PROGRAM G7_General
VAR_INPUT	SFCInit:BOOL;	END_VAR
VAR
	Memo_X_Precedent	:LREAL;	//Si plusieurs usinages au même X, pas besoin d'ouvrir et dég à chaque fois 
	Top_Cycles_Palp_Laser	:BOOL; //Lance le G7 des palpages buse et sommet du laser
	Fb_decode_real_Fct_M_: Fb_decode_real;
	Num_Unite_Cycle_Auto: INT;
	Num_operation_Cycle: INT;
	
	FE_Prepa_ISO_3D, FE_ISO_en_cours: F_trig;
	TON_ISO_en_cours, TON_Fin_Decoupe	:Ton;
	

END_VAR

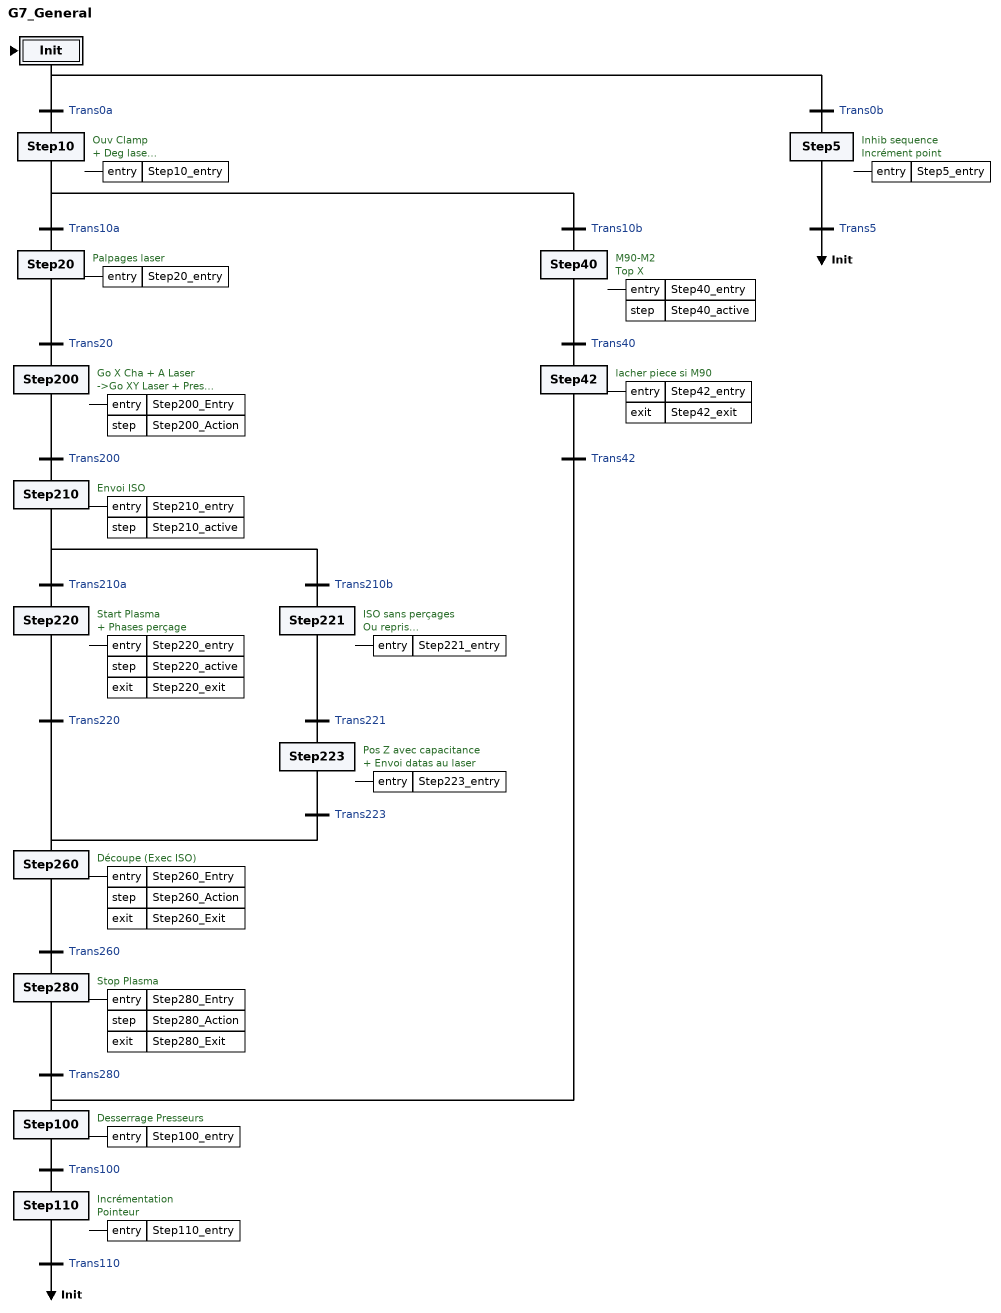
INITIAL_STEP Init:
END_STEP
TRANSITION FROM Init TO Step10
    := Trans0a;
END_TRANSITION
TRANSITION FROM Init TO Step5
    := Trans0b;
END_TRANSITION
// Inhib sequence
// Incrément point
STEP Step5:
    Step5_entry(P1);  // entry action
END_STEP
TRANSITION FROM Step5 TO Init
    := Trans5;
END_TRANSITION
// Ouv Clamp
// + Deg laser
// Si X Diff
// +Ctrl Palp Sommet
STEP Step10:
    Step10_entry(P1);  // entry action
END_STEP
TRANSITION FROM Step10 TO Step20
    := Trans10a;
END_TRANSITION
// Palpages laser
STEP Step20:
    Step20_entry(P1);  // entry action
END_STEP
TRANSITION FROM Step20 TO Step200
    := Trans20;
END_TRANSITION
// Go X Cha + A Laser
// ->Go XY Laser + Press
// +Prépa ISO
STEP Step200:
    Step200_Entry(P1);  // entry action
    Step200_Action(N);  // step action
END_STEP
TRANSITION FROM Step200 TO Step210
    := Trans200;
END_TRANSITION
// Envoi ISO
STEP Step210:
    Step210_entry(P1);  // entry action
    Step210_active(N);  // step action
END_STEP
TRANSITION FROM Step210 TO Step220
    := Trans210a;
END_TRANSITION
// Start Plasma
// + Phases perçage
STEP Step220:
    Step220_entry(P1);  // entry action
    Step220_active(N);  // step action
    Step220_exit(P0);  // exit action
END_STEP
TRANSITION FROM Step220 TO Step260
    := Trans220;
END_TRANSITION
TRANSITION FROM Step210 TO Step221
    := Trans210b;
END_TRANSITION
// ISO sans perçages
// Ou reprise
// Approche rapide Z laser
STEP Step221:
    Step221_entry(P1);  // entry action
END_STEP
TRANSITION FROM Step221 TO Step223
    := Trans221;
END_TRANSITION
// Pos Z avec capacitance
// + Envoi datas au laser
STEP Step223:
    Step223_entry(P1);  // entry action
END_STEP
TRANSITION FROM Step223 TO Step260
    := Trans223;
END_TRANSITION
// Découpe (Exec ISO)
STEP Step260:
    Step260_Entry(P1);  // entry action
    Step260_Action(N);  // step action
    Step260_Exit(P0);  // exit action
END_STEP
TRANSITION FROM Step260 TO Step280
    := Trans260;
END_TRANSITION
// Stop Plasma
STEP Step280:
    Step280_Entry(P1);  // entry action
    Step280_Action(N);  // step action
    Step280_Exit(P0);  // exit action
END_STEP
TRANSITION FROM Step280 TO Step100
    := Trans280;
END_TRANSITION
TRANSITION FROM Step10 TO Step40
    := Trans10b;
END_TRANSITION
// M90-M2
// Top X
STEP Step40:
    Step40_entry(P1);  // entry action
    Step40_active(N);  // step action
END_STEP
TRANSITION FROM Step40 TO Step42
    := Trans40;
END_TRANSITION
// lacher piece si M90
STEP Step42:
    Step42_entry(P1);  // entry action
    Step42_exit(P0);  // exit action
END_STEP
TRANSITION FROM Step42 TO Step100
    := Trans42;
END_TRANSITION
// Desserrage Presseurs
STEP Step100:
    Step100_entry(P1);  // entry action
END_STEP
TRANSITION FROM Step100 TO Step110
    := Trans100;
END_TRANSITION
// Incrémentation
// Pointeur
STEP Step110:
    Step110_entry(P1);  // entry action
END_STEP
TRANSITION FROM Step110 TO Init
    := Trans110;
END_TRANSITION

TRANSITION _tTrans210_1:
FE_Prepa_ISO_3D.Q
END_TRANSITION

ACTION Step10_entry:
IF Memo_X_Precedent <> Sequence[PT_Sequence].X THEN
 //Desserage presseur
  Presseur_Amont_K11.Dem_Desserrage:=
  Presseur_Aval_L12.Dem_Desserrage:=TRUE;
  Presseur_Amont_K11.Dem_Serrage:=
  Presseur_Aval_L12.Dem_Serrage:=FALSE;
 
 //Deg Z laser - Code M à voir
  IF Sequence[Pt_sequence].M<>50
  AND Sequence[Pt_sequence].M<>92
  AND Sequence[Pt_sequence].M<>93
  AND Sequence[Pt_sequence].M<>94
  AND NOT Deg_Laser_full_ok THEN
  	Top_deg_Laser_full:=TRUE; 
  END_IF
END_IF
 
// Contrôle palpage sommet
 IF Opt_Palp_Sommet_Tjs THEN	//On palpe tout le temps
 	Palpage_OK_Face_1 := Palpage_OK_Face_2 := FALSE;
 ELSIF Opt_Palp_Sommet_1Clamp THEN	// si début barre - donc seule la 1ere clamp dépassée - ou fin de barre - Fd de pince entre les 2 clamps - 
 	IF Sequence[Pt_sequence].X + Longueur_Barre_en_Pince <= Presseur_Aval_L12.Position_X
 		OR (Sequence[Pt_sequence].X >= Presseur_Amont_K11.Position_X AND Sequence[Pt_sequence].X < Presseur_Aval_L12.Position_X) THEN
 		Palpage_OK_Face_1 := Palpage_OK_Face_2 := FALSE;
 	ELSE
 		Palpage_OK_Face_1 := Palpage_OK_Face_2 := TRUE;
 	END_IF
 ELSE	//Si aucune des options de palpage, alors on ne palpe jamais
 	Palpage_OK_Face_1 := Palpage_OK_Face_2 := TRUE;
 END_IF

// Choix de la face d'usinage  
 IF Auto AND G7_Palpage_Sommet_L.Init.x THEN
 
 	(*Decodage des fonctions dans la sequence en cours*)
 	Fb_decode_real_Fct_M_(Valid:=TRUE,Real_Value:=Sequence[Pt_Sequence].M);
 	Num_Unite_Cycle_Auto:=Fb_decode_real_Fct_M_.Cent_Milliers;
 
 	Num_operation_Cycle:=LREAL_TO_INT(Sequence[Pt_Sequence].P10);
 	Decoupe := Num_operation_Cycle = 13;
 	Ecretage := Num_operation_Cycle = 15;
 
 	CASE Num_Unite_Cycle_Auto OF
 		1 : 	IF Decoupe THEN Face_Cible_Cycle := 1; END_IF;
 			IF Ecretage THEN Face_Cible_Cycle := 3; END_IF;	(* Normalement NON *)
 		2 : 	IF Decoupe THEN Face_Cible_Cycle := 2; END_IF;
 			IF Ecretage THEN Face_Cible_Cycle := 3; END_IF;
 	ELSE
 		Face_Cible_Cycle := 0;
 	END_CASE;
	
 END_IF;
END_ACTION

ACTION Step100_entry:
IF NOT X_Suivant_Idem THEN 
 Presseur_Amont_K11.Dem_Desserrage:=
 Presseur_Aval_L12.Dem_Desserrage:=TRUE;
 Presseur_Amont_K11.Dem_Serrage:=
 Presseur_Aval_L12.Dem_Serrage:=FALSE;
END_IF
END_ACTION

ACTION Step110_entry:
(*incrémentation pointeur*)
 Pt_Sequence:=Pt_Sequence+1;
END_ACTION

ACTION Step20_entry:
Top_Cycles_Palp_Laser:=true;
END_ACTION

ACTION Step200_Action:
IF En_pos_A_Laser AND Face_Cible=Face_En_Cours THEN
	//Laser
	 IF Reprise_decoupe THEN
	 	Pos_cible_X_Laser := Pnc_Start2[8];
	 	Pos_cible_Y_Laser := Pnc_Start2[9];
	 ELSE
		 //Gestion du Y selon la face en cours car impossible de juste changer le sens de comptage du Y 
		 IF Face_En_Cours=1 THEN // face réf, pas besoin de changer/adapter
	  		Pos_cible_Y_Laser := Sequence[Pt_Sequence].P2; //A changer des que comm dispo
		 ELSIF Face_En_Cours=2 THEN // face opp réf, Y + en montant donc inversion du Y. la côté reste la même, par contre attention lors du réglage de l'offset, aussi inversé : si besoin de descendre alors on augmente l'offset !
			Pos_cible_Y_Laser := -(Sequence[Pt_Sequence].P2); //A changer des que comm dispo
		 ELSIF Face_En_Cours=3 THEN	//Face écretage, je suppose que le driver envoie une cote = hauteur sommet - ep écrzetage. Pour cette position de face, Y laser compte en montant (s'éloignant de la réf)
			 Pos_cible_Y_Laser := Sequence[Pt_Sequence].P2 - Offset_Origine_Y_Laser;  
		 END_IF
	  	Pos_cible_X_Laser := Sequence[Pt_Sequence].P1; //A changer des que comm dispo
	 END_IF
	 En_pos_X_laser:=FALSE;
	 Top_X_laser	:=TRUE;
	 En_pos_Y_laser:=FALSE;
	 Top_Y_laser	:=TRUE;
	 
	//Presseurs
	Presseur_Amont_K11.Dem_Serrage:=
	Presseur_Aval_L12.Dem_Serrage:=TRUE;
	Presseur_Amont_K11.Dem_Desserrage:=
	Presseur_Aval_L12.Dem_Desserrage:=FALSE;
END_IF
END_ACTION

ACTION Step200_Entry:
// Positionnement chariot 
 Pos_cible_X:=Sequence[Pt_sequence].X;
 En_Pos_X:=FALSE;
 Top_X:=TRUE;
 
//Positionnement face laser
IF Face_Cible_Cycle <> 0 THEN
	Face_Cible 		:= Face_Cible_Cycle;
	Face_En_Pos 	:= FALSE;
	Top_Face 		:= TRUE;
END_IF;

(****************************** Prepa Fichier ISO ******************************)
(*Préparation fichier nc*)
Var_temp_rep_NC:=CONCAT(DINT_TO_STRING(LREAL_TO_DINT(Sequence[Pt_sequence].P7)),'.nc');

IF Reprise_decoupe THEN
	Var_temp_rep_NC:=CONCAT(DINT_TO_STRING(LREAL_TO_DINT(Sequence[Pt_sequence].P7)),'R.nc');
END_IF

Fichier_iso:=CONCAT(Repertoire_NC_Laser,Var_temp_rep_NC);
Start_ISO3D:=FALSE;
END_ACTION

ACTION Step210_active:
FE_Prepa_ISO_3D(clk := Prepa_ISO3D);
END_ACTION

ACTION Step210_entry:
FE_Prepa_ISO_3D(clk := FALSE);
Prepa_ISO3D := TRUE;
END_ACTION

ACTION Step220_active:
TON_Ecart_Pression_Gaz
(IN:=(ABS (LREAL_TO_INT(Consigne_Pression_Gaz) - Data14_Cutting_Gas_Pressure) > Ecart_Pression_Gaz) AND Tir_en_Cours AND Type_gaz = 0 ,
PT:=Tmps_Ecart_Pression);


IF TON_Ecart_Pression_Gaz.Q THEN Defaut_pression_gaz :=TRUE; END_IF
END_ACTION

ACTION Step220_entry:
(*Allumage torche*)
IF NOT Simul_decoupe AND NOT Bit_demo THEN
	Allumage_tete_laser:=TRUE;
END_IF
END_ACTION

ACTION Step220_exit:
TON_Ecart_Pression_Gaz(in:=false);
END_ACTION

ACTION Step221_entry:
Pos_cible_Z_Laser := pos_ref_torche - Tab_St_Recette_Laser[Index_Recette_Laser_Auto].Tb_Dec.Hauteur_Buse-Ep_secu;
En_pos_Z_Laser:=FALSE;
Top_Z_Laser:=TRUE;
END_ACTION

ACTION Step223_entry:
Pos_cible_Z_Laser := Pos_Reel_Z_Laser +( Prog_Capacitance_Actual_Value_mm -Tab_St_Recette_Laser[Index_Recette_Laser_Auto].Tb_Dec.Hauteur_Buse);
En_pos_Z_Laser:=FALSE;
Top_Z_Laser:=TRUE;

Consigne_Pression_Gaz					:=Tab_St_Recette_Laser[Index_Recette_Laser_Auto].Tb_dec.Pression_Gaz;
PLC_Prog_Power_Watt_Target					:=LREAL_TO_UDINT(Tab_St_Recette_Laser[Index_Recette_Laser_Auto].Tb_dec.Puissance_Laser);
PLC_Prog_Per_Cent_Of_Duty_Cycle_Target		:=LREAL_TO_UDINT(Tab_St_Recette_Laser[Index_Recette_Laser_Auto].Tb_dec.Duty_Cycle);
PLC_Prog_Frequency_0_20000Hz_Target			:=LREAL_TO_UDINT(Tab_St_Recette_Laser[Index_Recette_Laser_Auto].Tb_dec.Frequence_impulsion);
Prog_Distance_Focal_Demandee 			:=Tab_St_Recette_Laser[Index_Recette_Laser_Auto].Tb_dec.Distance_Focale;
Start_Gaz:=TRUE;
END_ACTION

ACTION Step260_Action:
FE_ISO_en_cours(clk:=ISO_en_cours);



TON_Ecart_Pression_Gaz
(IN:=(ABS (LREAL_TO_INT(Consigne_Pression_Gaz) - Data14_Cutting_Gas_Pressure) > Ecart_Pression_Gaz) AND Tir_Laser AND NOT F_M14 ,
PT:=Tmps_Ecart_Pression);


IF TON_Ecart_Pression_Gaz.Q THEN 
	Defaut_pression_gaz :=TRUE; 
END_IF
END_ACTION

ACTION Step260_Entry:
FE_ISO_en_cours(clk:=FALSE);
TON_ISO_en_cours(in:=FALSE);
(*Démarrage éxécution programme ISO*)

Start_ISO3D:=TRUE;
END_ACTION

ACTION Step260_Exit:
TON_ISO_en_cours(in:=FALSE);
(*Mise à jour "Séquence effectuée"*)
IF NOT Simul_decoupe THEN		(*Si reprise à faire sur 1 et 2 mais qu'on fait l'une puis l'autre alors il ne faut pas mettre à "ok" dès la 1e. Du coup, on ne met pas à "ok" après la 2e mais on s'en fout*)
	Sequence_status[Pt_sequence].Ok:=100;
END_IF

Asserv_Torche_On:=false;
END_ACTION

ACTION Step280_Action:
TON_fin_decoupe(in:=TRUE,pt:=T#500MS);

IF (Simul_decoupe OR Bit_demo) 
AND No_Move_Z_Laser AND NOT Z_Laser_en_mode_esclave
AND TON_fin_decoupe.Q AND NOT Top_deg_Laser_full THEN
	Top_deg_Laser_full:=TRUE;
END_IF
END_ACTION

ACTION Step280_Entry:
TON_fin_decoupe(in:=FALSE);
Allumage_tete_laser:=FALSE;
Tir_laser:=FALSE;
Start_ISO3D:=FALSE;
Start_Gaz:=FALSE;
END_ACTION

ACTION Step280_Exit:
TON_fin_decoupe(in:=FALSE);

(*Mise à jour Status sequence effectuée*)
Sequence_Status[Pt_Sequence].OK:=100;
END_ACTION

ACTION Step40_active:
IF Sequence[PT_Sequence].M=2 THEN
	IF Pos_reel_X < X_Cell_mesure_barre THEN
		Dem_Relevage_auto:=TRUE; //Compléter gestion pinces
	END_IF
END_IF
END_ACTION

ACTION Step40_entry:
Pos_Cible_X:=Sequence[Pt_Sequence].X;
En_pos_x:=FALSE;
Top_X:=TRUE;
END_ACTION

ACTION Step42_entry:
IF Sequence[PT_Sequence].M=90 THEN
	Dem_Serrage:=FALSE;
	Dem_Desserrage:=TRUE; //Compléter gestion pinces
END_IF
END_ACTION

ACTION Step42_exit:
Dem_Desserrage:=FALSE;

(*Mise à jour Status sequence effectuée*)
Sequence_Status[Pt_Sequence].OK:=100;
END_ACTION

ACTION Step5_entry:
Pt_sequence:=Pt_sequence+1;
END_ACTION

TRANSITION Trans0a:
TON_Auto.Q
AND	Sequence[Pt_Sequence].M<>0
AND	Sequence_Status[Pt_Sequence].OK=0

AND NOT Attente_Arret_Propre
END_TRANSITION

TRANSITION Trans0b:
(	Sequence[Pt_Sequence].M<>0
AND
	TON_Auto.Q
AND
	Sequence_Status[Pt_Sequence].OK=100)
	
AND NOT Attente_Arret_Propre //Si demande ouverture porte Laser
END_TRANSITION

TRANSITION Trans10:
Presseur_Amont_K11.Presseur_Haut
and Presseur_Aval_L12.Presseur_Haut
END_TRANSITION

TRANSITION Trans100:
(Presseur_Amont_K11.Presseur_Haut and Presseur_Aval_L12.Presseur_Haut) or X_Suivant_Idem
END_TRANSITION

TRANSITION Trans10a:
(Deg_Laser_full_ok
AND Presseur_Amont_K11.Presseur_Haut
AND Presseur_Aval_L12.Presseur_Haut) OR Memo_X_Precedent = Sequence[PT_Sequence].X
AND Decoupe OR Ecretage
END_TRANSITION

TRANSITION Trans10b:
(Deg_Laser_full_ok
AND Presseur_Amont_K11.Presseur_Haut
AND Presseur_Aval_L12.Presseur_Haut) 
AND Sequence[Pt_Sequence].M =90
OR Sequence[Pt_Sequence].M =2
END_TRANSITION

TRANSITION Trans110:
step110.t>T#20ms
END_TRANSITION

TRANSITION Trans20:
G7_Master_Palpages.Init.x
AND (NOT Nv_ProcessID AND Prog_Capacitance_Calibration_OK)
AND (Palpage_OK_Face_1 AND Palpage_OK_Face_2)
END_TRANSITION

TRANSITION Trans200:
//Axes en pos
En_pos_X AND NOT Top_X
AND En_pos_X_Laser AND NOT Top_X_Laser
AND	En_pos_Y_Laser AND NOT Top_Y_Laser
AND En_pos_Z_Laser AND NOT Top_Z_Laser
AND En_pos_A_Laser AND NOT Top_A_Laser
//Presseurs en place
AND Presseur_Amont_K11.Presseur_EnPlace
AND Presseur_Aval_L12.Presseur_EnPlace

AND 
	Sequence[Pt_sequence].P26=Pnc_Laser[20]
	
AND step200.t>T#20MS
END_TRANSITION

TRANSITION Trans210a:
FE_Prepa_ISO_3D.Q 
AND Tab_St_Recette_Laser[Index_Recette_Laser_Auto].Tb_Perc[1].Puissance_Laser <>0 // La 1ère phase de perçage existe, donc il y a bien au moins une phase de perçage
AND NOT Reprise_decoupe
END_TRANSITION

TRANSITION Trans210b:
FE_Prepa_ISO_3D.Q 
AND Tab_St_Recette_Laser[Index_Recette_Laser_Auto].Tb_Perc[1].Puissance_Laser=0	//Pas de phase de perçage
or Reprise_decoupe
END_TRANSITION

TRANSITION Trans220:
(*Signal arc amorcé venant de la source, après les phases de perçages  *)


(*Découpe laser*)

	(	Sequence[Pt_sequence].P1=0
	AND
	(*Torche 1*)
		((Laser_ok_pour_decoupe AND G7_Cycle_Percages_Laser.Step31.x)				(*Machine à 1:		Cas normal:					arc 1 transféré et Pierce Delay écoulé*)
		OR Simul_decoupe AND G7_Cycle_Percages_Laser.Init.x							(*Machine à 1:		Simulation de découpe:		on n'a pas allumé la torche 1 alors faut bien passer*)
		OR (Bit_demo))) //AND NOT Option_lifter_plasma_VB)							(*Machine à 1:		Mode démo:					on n'a pas allumé la torche 1 alors faut bien passer*)
END_TRANSITION

TRANSITION Trans221:
step221.t>T#20MS
AND En_pos_Z_Laser
and not Top_Z_Laser
END_TRANSITION

TRANSITION Trans223:
step223.t>T#20MS
AND ABS(Prog_Capacitance_Actual_Value_mm -Tab_St_Recette_Laser[Index_Recette_Laser_Auto].Tb_Dec.Hauteur_Buse) <0.5
AND Data13_Cutting_Gas_Temp			=	Consigne_Pression_Gaz	AND 			
_1_LASER.Feedback_Laser_Power	=	PLC_Prog_Power_Watt_Target	AND 		
_1_LASER.Feedback_Laser_Duty	=	PLC_Prog_Per_Cent_Of_Duty_Cycle_Target AND	
_1_LASER.Feedback_Laser_Freq	=	PLC_Prog_Frequency_0_20000Hz_Target AND		
Prog_Distance_Focal_Reelle 		= 	Prog_Distance_Focal_Demandee
END_TRANSITION

TRANSITION Trans260:
(*Attente fin d'éxécution programme ISO*)
FE_ISO_en_cours.Q
END_TRANSITION

TRANSITION Trans280:
	X_no_move
AND
	TON_fin_decoupe.Q
AND
	(NOT Simul_decoupe
	OR
	(Simul_decoupe
	AND Bp_Depart_Cycle))	(*Ne surtout pas supprimer cette attente DCY en simul (+MessOp.txt), car risque de ne jamais découper les pièces simulées*)
AND
//	(NOT Bit_demo
//	OR
//	(Bit_demo
//	AND 
	Deg_Laser_full_ok
//	))
END_TRANSITION

TRANSITION Trans40:
En_Pos_X
and not Top_X
END_TRANSITION

TRANSITION Trans42:
Fin_Desserage_Pince or Sequence[Pt_Sequence].M=2
END_TRANSITION

TRANSITION Trans5:
true
END_TRANSITION

END_PROGRAM

(* stored: Version 1.1.0.1
   POU G7_General: Id {5f9f3406-b176-444b-8d98-626ce3907be7}, SpecialFunc None
   Transition _tTrans210_1: Id {3fac5508-bcbc-4a34-932a-bd11aa626656}
   Action Step10_entry: Id {bb8ddf34-7b46-4d2a-bb0f-9493f70d6a20}
   Action Step100_entry: Id {93586d4c-e79e-4084-9e9e-bc2b656c8645}
   Action Step110_entry: Id {e7b29dd0-e6be-4f66-9626-84fb78622d04}
   Action Step20_entry: Id {9dbf7d81-53b6-4ac1-8a2a-dd36ba0e5023}
   Action Step200_Action: Id {a514a9cd-791b-4703-b1a6-01074b7c77f3}
   Action Step200_Entry: Id {1779b138-bc46-448d-89f6-71c3648c2cc1}
   Action Step210_active: Id {4e8ea5b6-c17b-45b6-9942-9206653e17ac}
   Action Step210_entry: Id {c1be57c6-1102-4390-bc96-edd366469950}
   Action Step220_active: Id {9d98ecdf-fcb4-420c-b88f-8132c706f74f}
   Action Step220_entry: Id {7aaf9abd-0999-45c6-83be-75d8967a2d85}
   Action Step220_exit: Id {98b4d34f-b157-4045-8d74-512afd97bea2}
   Action Step221_entry: Id {136b9709-3735-4173-9f23-c7d57741e24c}
   Action Step223_entry: Id {8280820c-8759-470a-b7f0-98ca53832f93}
   Action Step260_Action: Id {47d2b299-c154-4f53-a0b3-9eef55b28759}
   Action Step260_Entry: Id {f163747f-7ec1-408b-8132-487fa5ad8d91}
   Action Step260_Exit: Id {769d3bf1-7230-4a0f-8755-01bdc63b7777}
   Action Step280_Action: Id {61e837ea-74c2-4ba4-ae56-849852214210}
   Action Step280_Entry: Id {d9ba3964-249d-4eab-90c7-2bb5530741af}
   Action Step280_Exit: Id {4b93cf75-66f8-457b-a23a-2b5bd36aaf94}
   Action Step40_active: Id {dc75d40f-8215-4159-b504-7b2d64d20ef3}
   Action Step40_entry: Id {fd00367a-e3c8-46e7-8c42-847f0ce72a98}
   Action Step42_entry: Id {612d719a-e90d-43db-a655-05c22e08119d}
   Action Step42_exit: Id {2d37d738-63cb-44c8-8c1e-de0bb8a39c85}
   Action Step5_entry: Id {474fd148-0a04-4e74-9fe5-cf9fd26feb7f}
   Transition Trans0a: Id {dda23c8e-c927-4285-896f-d7a2ad0d4a2d}
   Transition Trans0b: Id {e155ca35-c358-456b-8b4b-b0f5b65dd783}
   Transition Trans10: Id {694feb76-9865-4a22-b134-b54f1d0938f6}
   Transition Trans100: Id {5b3d41cc-9a93-417f-83c3-cbceaa1e9e3b}
   Transition Trans10a: Id {bdd53c74-e5db-49fd-8d60-cb7893b310fb}
   Transition Trans10b: Id {38c658e5-2377-4d01-9006-11a08ea633aa}
   Transition Trans110: Id {c1145a46-2412-497c-aacb-ac426331fbc7}
   Transition Trans20: Id {fab8237b-cf37-4cd7-87be-419e62b023dc}
   Transition Trans200: Id {22e3c04d-1447-47b5-b07f-58062277d9a2}
   Transition Trans210a: Id {bc5b8177-fb42-4a83-ab52-0d64ff904a7c}
   Transition Trans210b: Id {13faeb58-343f-4fab-be0b-91c1daad5107}
   Transition Trans220: Id {3bea94e6-fe6b-417e-b3be-70f1d5cb1342}
   Transition Trans221: Id {c8eb0901-8278-40e2-95aa-286df6b1b1f2}
   Transition Trans223: Id {ce3d769d-61b5-4e24-9e53-7de6cba5017c}
   Transition Trans260: Id {e571c51e-ee71-46a5-bd1e-0a6504be934f}
   Transition Trans280: Id {dad065d7-8c01-450e-b84e-1b00f86c56fc}
   Transition Trans40: Id {57c2974c-58f9-4f76-8ce8-e2dc0eb0a864}
   Transition Trans42: Id {0b5ace2a-c1d8-420a-be6b-d29467fd1b27}
   Transition Trans5: Id {0fac0bc7-f62d-43f7-b714-d7592de94d68} *)
